ABB RobotStudio station: Linea_ensamblaje_A3.rsstn

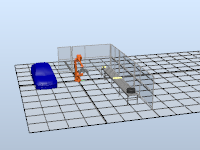
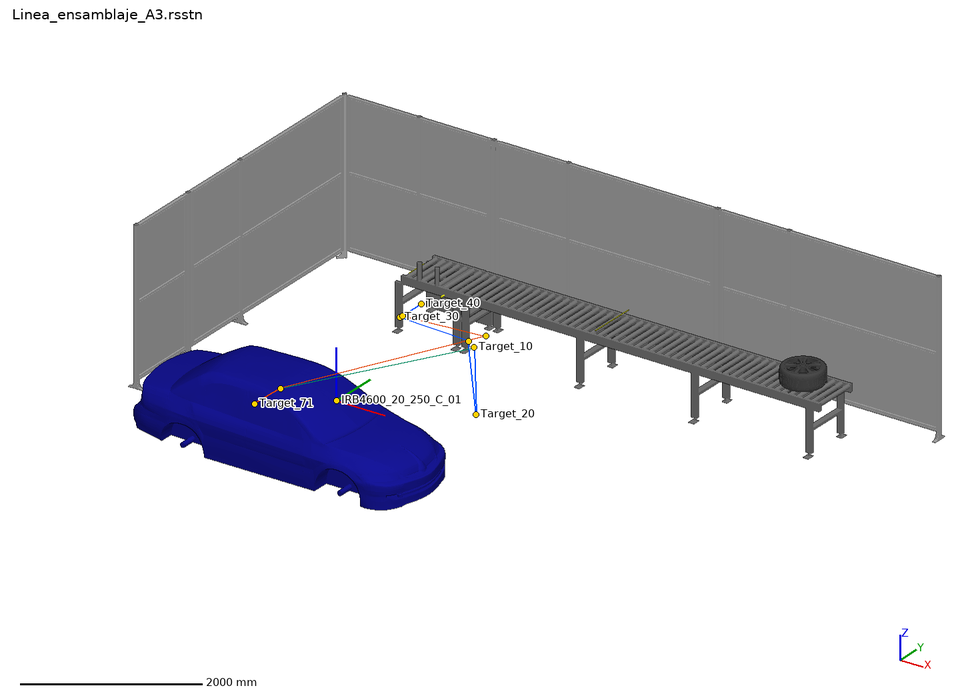
[picture v1: parts stored in the station drawn from their meshes, with robot base, taught points and paths (robot models come from the ABB library and are not in the file)]
Station Línea de ensamblaje v5 (saved by RobotStudio 21.2.9526.0)
Controller Controlador
  mechanical unit ROB_1: IRB4600_20_250_C_01, 6 joints, base frame (0, 0, 0) mm
Layout (positions relative to the parent item):
  - Carroceria [part] at (3000, -2500, 500) mm, rotated rx 90 ry 0 rz 90 deg, size 1363.4 x 983.1 x 3612.1 mm
  - Rueda banda [part] at (4754.35, 2138.13, 907.94) mm, rotated rx -11.7 ry -90 rz 47.69 deg, size 228.1 x 532.2 x 532.2 mm
  - lancerwheel_3 [part] at (2126.39, -1779.96, 250) mm, rotated rx 0 ry 0 rz 90 deg, size 223.1 x 527.9 x 528 mm
  - Banda [part] at (0, 300, 0) mm, size 4904.4 x 741.5 x 692.3 mm
  - Logica_Banda [smart component]
      signals: DO AcercarGripper, DI RotarMesaOriginal
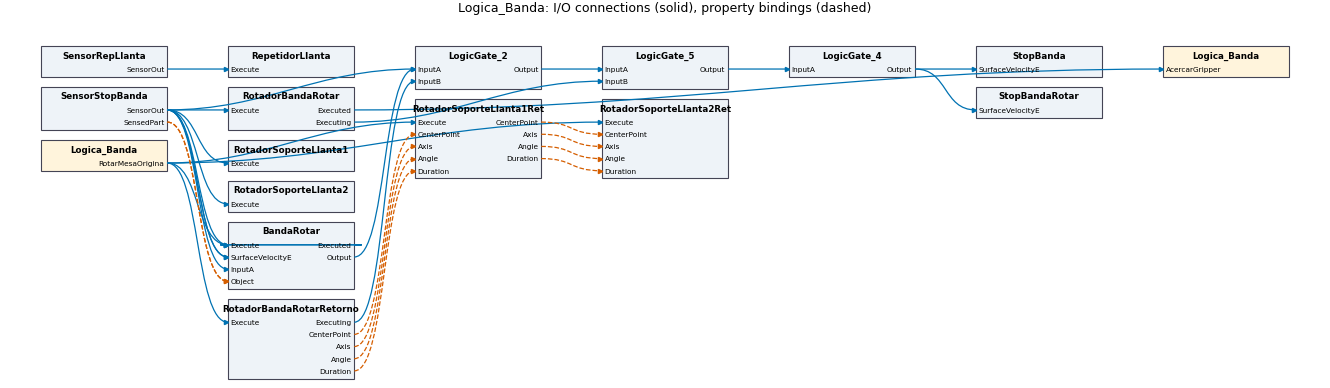
      connections:
        SensorRepLlanta.SensorOut -> RepetidorLlanta.Execute
        BandaRotar.Executed -> BandaRotar2.Execute
        BandaRotar2.Executed -> BandaRotar3.Execute
        SensorStopBanda.SensorOut -> PhysicsControl.SurfaceVelocityEnabled
        SensorStopBanda.SensorOut -> LinearMover2.Execute
        SensorStopBanda.SensorOut -> PhysicsControl_3.SurfaceVelocityEnabled
        RotadorBandaRotar.Executed -> Logica_Banda.AcercarGripper
        Logica_Banda.RotarMesaOriginal -> Rotator2.Execute
        Logica_Banda.RotarMesaOriginal -> RotadorBandaRotarRetorno.Execute
        Logica_Banda.RotarMesaOriginal -> RotadorSoporteLlanta1Ret.Execute
        Logica_Banda.RotarMesaOriginal -> RotadorSoporteLlanta2Ret.Execute
        SensorStopBanda.SensorOut -> LogicGate.InputA
        SensorStopBanda.SensorOut -> RotadorBandaRotar.Execute
        SensorStopBanda.SensorOut -> RotadorSoporteLlanta1.Execute
        SensorStopBanda.SensorOut -> RotadorSoporteLlanta2.Execute
        LogicGate.Output -> LogicGate_2.InputA
        LogicGate_4.Output -> StopBanda.SurfaceVelocityEnabled
        LogicGate_4.Output -> StopBandaRotar.SurfaceVelocityEnabled
        RotadorBandaRotarRetorno.Executing -> LogicGate_2.InputB
        SensorStopBanda.SensorOut -> LogicGate_2.InputA
        LogicGate_2.Output -> LogicGate_5.InputA
        RotadorBandaRotar.Executing -> LogicGate_5.InputB
        LogicGate_5.Output -> LogicGate_4.InputA
        SensorStopBanda.SensedPart => LinearMover2.Object
        SensorStopBanda.SensedPart => PhysicsControl_3.Object
        RotadorBandaRotarRetorno.CenterPoint => RotadorSoporteLlanta1Ret.CenterPoint
        RotadorSoporteLlanta1Ret.CenterPoint => RotadorSoporteLlanta2Ret.CenterPoint
        RotadorBandaRotarRetorno.Axis => RotadorSoporteLlanta1Ret.Axis
        RotadorSoporteLlanta1Ret.Axis => RotadorSoporteLlanta2Ret.Axis
        RotadorBandaRotarRetorno.Angle => RotadorSoporteLlanta1Ret.Angle
        RotadorSoporteLlanta1Ret.Angle => RotadorSoporteLlanta2Ret.Angle
        RotadorBandaRotarRetorno.Duration => RotadorSoporteLlanta1Ret.Duration
        RotadorSoporteLlanta1Ret.Duration => RotadorSoporteLlanta2Ret.Duration
    - SensorRepLlanta [smart component, from Components\LineSensor.rslib] at (-3000, 300, 54.91) mm
        properties: Start=[5.191342 2.154215 0.686]; End=[5.18975 1.521334 0.686]; Radius=0.005; SensedPart=(none); SensedPoint=[0 0 0]
      - _sensorPart_ [part], size 11.6 x 632.9 x 10 mm
    - RepetidorLlanta [smart component, from Components\Source.rslib]
        properties: Source=Rueda banda; Copy=(none); Parent=(none); Position=[5.098082 2.13994 0.97376]; Orientation=[0 -1.5707963267949 0]; Transient=true; PhysicsBehavior=3
    - SensorStopBanda [smart component, from Components\LineSensor.rslib] at (0, 300, 0) mm
        properties: Start=[-0.3 1.80049 0.75]; End=[-0.3 1.516713 0.75]; Radius=0.005; SensedPart=(none); SensedPoint=[0 0 0]
      - _sensorPart_ [part], size 10 x 283.8 x 10 mm
    - StopBanda [smart component, from Components\PhysicsControl.rslib] at (-0.51, 167.85, 24.33) mm
        properties: Object=Banda; Behavior=1; SurfaceVelocity=0.3
    - RotadorBandaRotar [smart component, from Components\Rotator2.rslib]
        properties: Object=Bandamovil1; CenterPoint=[-0.107807 2.133495 0.496844]; Axis=[1 0 0]; Angle=1.5707963267949; Duration=2; Reference=Global; ReferenceObject=(none)
    - StopBandaRotar [smart component, from Components\PhysicsControl.rslib]
        properties: Object=Bandamovil1; Behavior=2; SurfaceVelocity=0.3
    - RotadorSoporteLlanta1 [smart component, from Components\Rotator2.rslib]
        properties: Object=SoporteLlanta1; CenterPoint=[-0.107807 2.133495 0.496844]; Axis=[1 0 0]; Angle=1.5707963267949; Duration=2; Reference=Global; ReferenceObject=(none)
    - RotadorSoporteLlanta2 [smart component, from Components\Rotator2.rslib]
        properties: Object=SoporteLlanta2; CenterPoint=[-0.107807 2.133495 0.496844]; Axis=[1 0 0]; Angle=1.5707963267949; Duration=2; Reference=Global; ReferenceObject=(none)
    - RotadorBandaRotarRetorno [smart component, from Components\Rotator2.rslib]
        properties: Object=Bandamovil1; CenterPoint=[-0.107807 2.133495 0.496844]; Axis=[1 0 0]; Angle=-1.5707963267949; Duration=2; Reference=Global; ReferenceObject=(none)
    - RotadorSoporteLlanta2Ret [smart component, from Components\Rotator2.rslib]
        properties: Object=SoporteLlanta2; CenterPoint=[-0.107807 2.133495 0.496844]; Axis=[1 0 0]; Angle=-1.5707963267949; Duration=2; Reference=Global; ReferenceObject=(none)
    - RotadorSoporteLlanta1Ret [smart component, from Components\Rotator2.rslib]
        properties: Object=SoporteLlanta1; CenterPoint=[-0.107807 2.133495 0.496844]; Axis=[1 0 0]; Angle=-1.5707963267949; Duration=2; Reference=Global; ReferenceObject=(none)
    - LogicGate_2 [smart component, from Components\LogicGate.rslib]
        properties: Operator=OR; Delay=0
    - LogicGate_4 [smart component, from Components\LogicGate.rslib]
        properties: Operator=NOT; Delay=0
    - LogicGate_5 [smart component, from Components\LogicGate.rslib]
        properties: Operator=OR; Delay=0
  - Bandamovil1 [part] at (-107.84, 2133.21, 496.61) mm, size 696.4 x 640.5 x 227.8 mm
  - Bandamovil2 [part] at (-63.61, 2138.31, 496.25) mm, rotated rx 90 ry 0 rz 90 deg, size 742.4 x 599.6 x 864.8 mm
  - SoporteLlanta1 [part] at (-180.93, 1841.31, 794.89) mm, size 59.4 x 59.4 x 223.5 mm
  - SoporteLlanta2 [part] at (55.93, 1841.31, 794.89) mm, size 59.4 x 59.4 x 223.5 mm
  - GripperRueda_2 [mechanism, from Gripper\GripperRueda.rslib] at (1406.98, 0, 1354.03) mm, rotated rx 178.86 ry 0 rz -90 deg; joint values [0, 0, 0] (rad or m)
  - IRB4600_20_250_C_01 [mechanism, from Robots\IRB4600_20_250_C_01.rslib] at (0, 0, 0) mm; joint values [0, 0, 0.2631, 0, 1.3277, -1.5708] (rad or m)
  - Logica_Gripper [smart component]
      signals: DI CierraGripper, DI AbreGripper
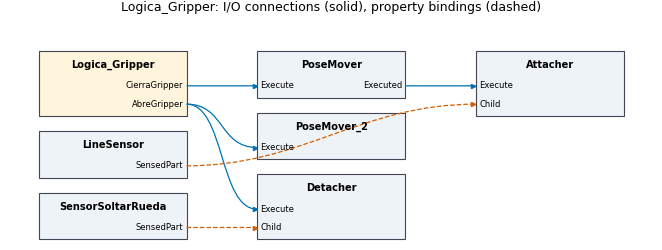
      connections:
        Logica_Gripper.CierraGripper -> PoseMover.Execute
        PoseMover.Executed -> Attacher.Execute
        Logica_Gripper.AbreGripper -> Detacher.Execute
        Logica_Gripper.AbreGripper -> PoseMover_2.Execute
        LineSensor.SensedPart => Attacher.Child
        SensorSoltarRueda.SensedPart => Detacher.Child
    - PoseMover [smart component, from Components\PoseMover.rslib]
        properties: Mechanism=GripperRueda_2; Pose=2; Duration=0.2
    - Attacher [smart component, from Components\Attacher.rslib]
        properties: Parent=GripperRueda_2; Flange=0; Child=Rueda banda; Mount=false; Offset=[0 0 0]; Orientation=[0 0 0]
    - LineSensor [smart component, from Components\LineSensor.rslib] at (-107.84, 2133.73, 496.56) mm, rotated rx 90 ry 0 rz 0 deg
        properties: Start=[0.278167 0.111436 0.268002999999999]; End=[0.272931 0.111436 0.372674999999999]; Radius=0.01; SensedPart=Rueda banda; SensedPoint=[0.170324996948242 1.86573095703125 0.608]
      - _sensorPart_ [part], size 25.2 x 20 x 105.7 mm
    - Detacher [smart component, from Components\Detacher.rslib]
        properties: Child=(none); KeepPosition=true
    - PoseMover_2 [smart component, from Components\PoseMover.rslib]
        properties: Mechanism=GripperRueda_2; Pose=3; Duration=0.2
    - SensorSoltarRueda [smart component, from Components\LineSensor.rslib] at (0, -1455.8, 0) mm
        properties: Start=[0.26 -0.444199968527614 0.474]; End=[0.26 -0.344199968527614 0.474]; Radius=0.005; SensedPart=(none); SensedPoint=[0 0 0]
      - _sensorPart_ [part], size 10 x 100 x 10 mm
  - Fence [graphiccomponentgroup]
    - Segment 1 [part], size 44.1 x 184.1 x 2000 mm
    - Segment 2 [part], size 2022 x 184.1 x 2000 mm
    - Segment 2 [part], size 980.6 x 184 x 2000 mm
    - Segment 3 [part], size 2000 x 184 x 2000 mm
    - Segment 3 [part], size 1019.2 x 184 x 2000 mm
    - Segment 4 [part], size 1004 x 184 x 2000 mm
    - Segment 4 [part], size 1083.2 x 158.4 x 2000 mm
    - Segment 5 [part], size 184.1 x 2000 x 2000 mm
    - Segment 5 [part], size 184.1 x 1023 x 2000 mm
    - Segment 6 [part], size 184.1 x 995 x 2000 mm
Attachment: GripperRueda_2 is attached to IRB4600_20_250_C_01 / Link6
Attachment: LineSensor is attached to Bandamovil1
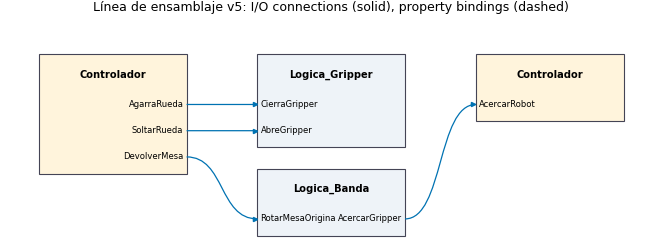
Station logic (signal -> signal, property => property):
  Logica_Banda.AcercarGripper -> Controlador.AcercarRobot
  Controlador.AgarraRueda -> Logica_Gripper.CierraGripper
  Controlador.SoltarRueda -> Logica_Gripper.AbreGripper
  Controlador.DevolverMesa -> Logica_Banda.RotarMesaOriginal
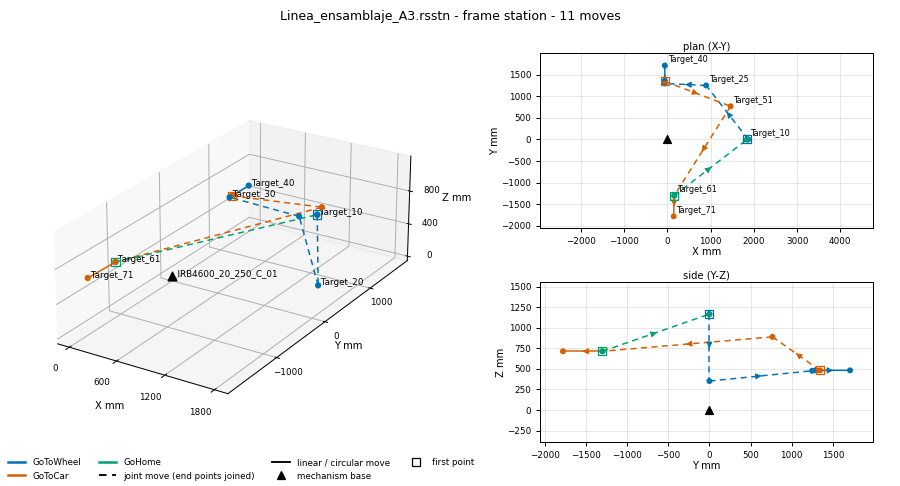
[picture p0: tool path of Linea_ensamblaje_A3.rsstn in frame station, 11 of 11 moves have a stored position in this frame; points joined in program order, loops and branches not executed]
Targets, tools, work objects and paths stored in the station, written as RAPID:
! task T_ROB1
MODULE CalibData
  PERS tooldata GripperRueda_1:=[TRUE,[[0,-442,180],[0.5,0.5,-0.5,0.5]],[1,[0,8,0],[1,0,0,0],0,0,0]];
  TASK PERS wobjdata Workobject_1:=[FALSE,TRUE,"",[[0,0,0],[1,0,0,0]],[[0,0,0],[1,0,0,0]]];
  PERS tooldata Tooldata_1:=[TRUE,[[0,-442,180],[0.5,0.5,-0.5,0.5]],[1,[0,8,0],[1,0,0,0],0,0,0]];
ENDMODULE

! task T_ROB1
MODULE Module1
  CONST robtarget Target_30:=[[-59.962976648,1292.993835357,482.280295667],[0.502544841,-0.497475013,0.503471471,0.496471321],[1,0,-1,0],[9E+09,9E+09,9E+09,9E+09,9E+09,9E+09]];
  CONST robtarget Target_20:=[[1869.841482343,0,351.982794242],[0.708176688,0,0.706035253,0],[0,0,-1,0],[9E+09,9E+09,9E+09,9E+09,9E+09,9E+09]];
  CONST robtarget Target_10:=[[1845.310568624,0,1165.263528275],[0.700028676,0,0.714114734,0],[0,0,-2,0],[9E+09,9E+09,9E+09,9E+09,9E+09,9E+09]];
  CONST robtarget Target_41:=[[-58.57494655,1343.92028614,482.058366266],[0.502544841,-0.497475013,0.503471471,0.496471321],[1,0,-1,0],[9E+09,9E+09,9E+09,9E+09,9E+09,9E+09]];
  CONST robtarget Target_25:=[[895.494158417,1248.976757634,476.638064362],[0.634915636,-0.311287272,0.634852453,0.311359492],[0,0,-1,0],[9E+09,9E+09,9E+09,9E+09,9E+09,9E+09]];
  CONST robtarget Target_40:=[[-58.57494655,1709.225040825,482.058366266],[0.502544841,-0.497475013,0.503471471,0.496471321],[1,0,-1,0],[9E+09,9E+09,9E+09,9E+09,9E+09,9E+09]];
  CONST robtarget Target_51:=[[1461.868533648,766.758695219,889.042973148],[0.776683991,-0.185116689,0.577593438,0.169940022],[0,-1,-1,0],[9E+09,9E+09,9E+09,9E+09,9E+09,9E+09]];
  CONST robtarget Target_61:=[[158.985392675,-1299.630065486,713.888752887],[0.51321887,0.490480502,0.506512222,-0.489367589],[-1,0,-1,0],[9E+09,9E+09,9E+09,9E+09,9E+09,9E+09]];
  CONST robtarget Target_71:=[[145.32624319,-1779.204024326,713.888504299],[0.505128934,0.498716509,0.498405113,-0.49771372],[-1,0,-1,0],[9E+09,9E+09,9E+09,9E+09,9E+09,9E+09]];
  PROC GoToWheel()
    MoveJ Target_10,v1500,z1,Tooldata_1\WObj:=Workobject_1;
    MoveJ Target_20,v1500,z1,Tooldata_1\WObj:=Workobject_1;
    MoveJ Target_25,v1500,z1,Tooldata_1\WObj:=Workobject_1;
    MoveJ Target_30,v1500,z1,Tooldata_1\WObj:=Workobject_1;
    WaitDI AcercarRobot,1;
    MoveL Target_40,v200,fine,GripperRueda_1\WObj:=Workobject_1;
    SetDO AgarraRueda,1;
    WaitTime 1;
    SetDO AgarraRueda,0;
  ENDPROC
  PROC main()
    SetDO DevolverMesa,0;
    GoToWheel;
    GoToCar;
    GoHome;
    main;
  ENDPROC
  PROC GoToCar()
    MoveJ Target_41,v1500,z1,Tooldata_1\WObj:=Workobject_1;
    MoveJ Target_51,v1500,z1,Tooldata_1\WObj:=Workobject_1;
    MoveJ Target_61,v1500,z1,Tooldata_1\WObj:=Workobject_1;
    MoveL Target_71,v200,fine,Tooldata_1\WObj:=Workobject_1;
    SetDO SoltarRueda,1;
    WaitTime 1;
    SetDO SoltarRueda,0;
  ENDPROC
  PROC GoHome()
    MoveL Target_61,v200,fine,Tooldata_1\WObj:=Workobject_1;
    MoveJ Target_10,v1500,z1,Tooldata_1\WObj:=Workobject_1;
    SetDO DevolverMesa,1;
  ENDPROC
ENDMODULE

